// TIA Portal project "4_side_traffic_light_real_clock" (V16)

(* hardware
DEVICE "S7-1200 station_1"  S7-1200 Station
   slot 0: "Rack_0"  S7-1200 Rack  Rack  V1.0
   slot 1: "PLC_1"  CPU 1212C DC/DC/DC  6ES7 212-1AE40-0XB0  V4.4
*)

// ===== PLC "PLC_1"  CPU 1212C DC/DC/DC =====

VAR_GLOBAL   // PLC tag table "Default tag table"
   "Tag_1" AT %M0.0 : Bool;
   "Tag_2" AT %M0.1 : Bool;
   "Tag_3" AT %M0.2 : Bool;
   "green1" AT %Q0.0 : Bool;
   "green2" AT %Q0.1 : Bool;
   "green3" AT %Q0.2 : Bool;
   "green4" AT %Q0.3 : Bool;
   "yellow1" AT %Q0.4 : Bool;
   "yellow2" AT %Q0.5 : Bool;
   "yellow3" AT %Q0.6 : Bool;
   "yellow4" AT %Q0.7 : Bool;
   "red1" AT %Q1.0 : Bool;
   "red2" AT %Q1.1 : Bool;
   "red3" AT %Q1.2 : Bool;
   "red4" AT %Q1.3 : Bool;
   "emergency1" AT %M1.2 : Bool;
   "emergency2" AT %M1.3 : Bool;
   "emergency3" AT %M1.4 : Bool;
   "emergency4" AT %M1.5 : Bool;
   "set date and time" AT %M9.0 : Bool;
   "night mode" AT %M4.3 : Bool;
   "yellow blinker" AT %Q1.6 : Bool;
END_VAR

DATA_BLOCK "read data block"   // DB2
{ S7_Optimized_Access := 'TRUE' }
VERSION : 0.1
   VAR
      "read data block" : DTL;
      status : Int;
   END_VAR
BEGIN
END_DATA_BLOCK

DATA_BLOCK "write data block"   // DB3
{ S7_Optimized_Access := 'TRUE' }
VERSION : 0.1
   VAR
      "write data block" : DTL;
      status : Int;
   END_VAR
BEGIN
END_DATA_BLOCK

// folder: System blocks/Program resources

DATA_BLOCK "timer1"   // DB1
{ S7_Optimized_Access := 'TRUE' }
AUTHOR : Simatic
FAMILY : IEC
NAME : IEC_TMR
VERSION : 1.0
// stored: InstanceOfName IEC_TIMER
"IEC_TIMER"
BEGIN
END_DATA_BLOCK

DATA_BLOCK "timer2"   // DB4
{ S7_Optimized_Access := 'TRUE' }
AUTHOR : Simatic
FAMILY : IEC
NAME : IEC_TMR
VERSION : 1.0
// stored: InstanceOfName IEC_TIMER
"IEC_TIMER"
BEGIN
END_DATA_BLOCK

DATA_BLOCK "timer3"   // DB5
{ S7_Optimized_Access := 'TRUE' }
AUTHOR : Simatic
FAMILY : IEC
NAME : IEC_TMR
VERSION : 1.0
// stored: InstanceOfName IEC_TIMER
"IEC_TIMER"
BEGIN
END_DATA_BLOCK

// folder: (top level)

ORGANIZATION_BLOCK "Main"   // OB1, LAD, ProgramCycle
TITLE = "Main Program Sweep (Cycle)"
{ S7_Optimized_Access := 'TRUE' }
VERSION : 0.1
   VAR_INPUT
      Initial_Call : Bool;   // Initial call of this OB
      Remanence : Bool;   // =True, if remanent data are available
   END_VAR
BEGIN

REGION Network 1
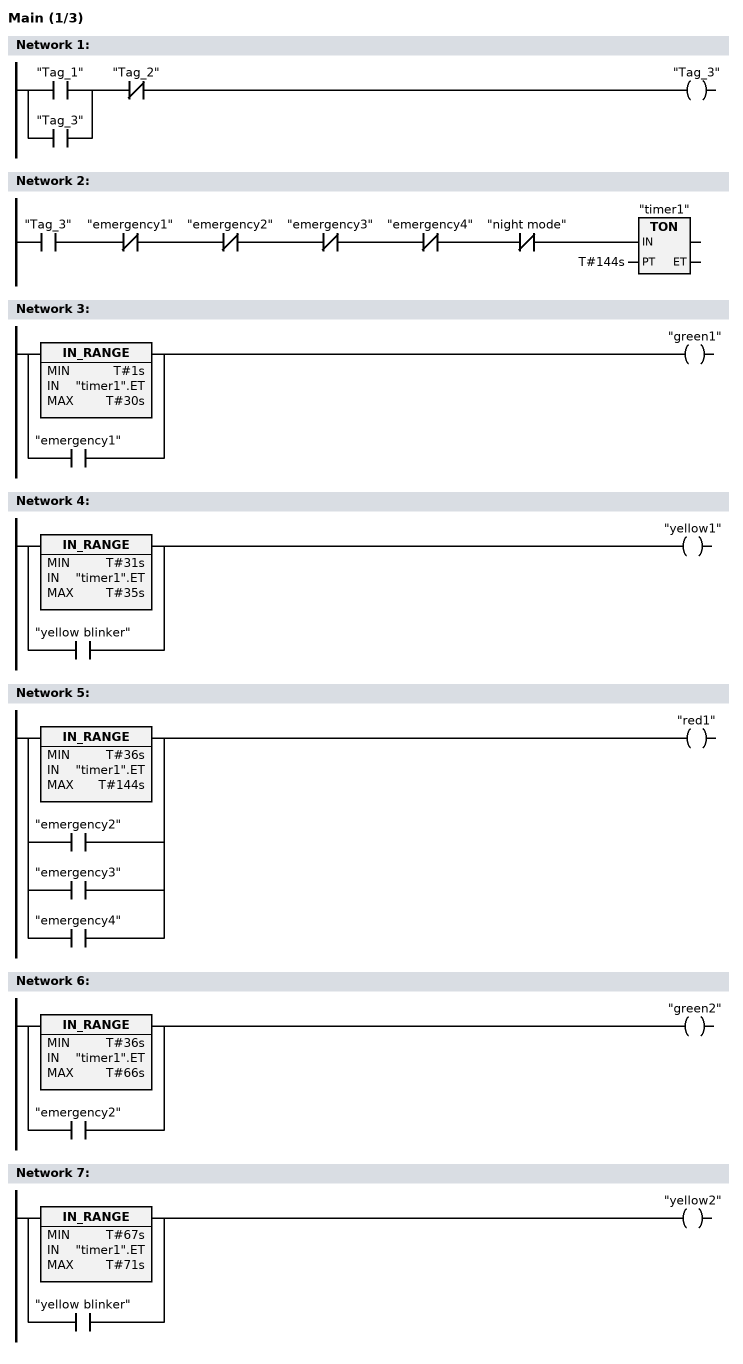
   RUNG wire#powerrail
      Contact( "Tag_1" )
      wire#w1
      I_Contact( "Tag_2" )
      Coil( "Tag_3" )
   END_RUNG
   RUNG wire#powerrail
      Contact( "Tag_3" )
   END_RUNG wire#w1
   // the same network as SCL:
   "Tag_3" := ("Tag_1" OR "Tag_3") AND NOT "Tag_2";
END_REGION

REGION Network 2
   "timer1".TON(IN := "Tag_3" AND NOT "emergency1" AND NOT "emergency2" AND NOT "emergency3" AND NOT "emergency4" AND NOT "night mode",
                PT := T#144s);
END_REGION

REGION Network 3
   RUNG wire#powerrail
      { S7_Templates := "SrcType := DInt" } InRange(min := T#1s, in := "timer1".ET, max := T#30s)
      wire#w1
      Coil( "green1" )
   END_RUNG
   RUNG wire#powerrail
      Contact( "emergency1" )
   END_RUNG wire#w1
   // the same network as SCL:
   "green1" := ((T#1s <= "timer1".ET) AND ("timer1".ET <= T#30s)) OR "emergency1";
END_REGION

REGION Network 4
   RUNG wire#powerrail
      { S7_Templates := "SrcType := DInt" } InRange(min := T#31s, in := "timer1".ET, max := T#35s)
      wire#w1
      Coil( "yellow1" )
   END_RUNG
   RUNG wire#powerrail
      Contact( "yellow blinker" )
   END_RUNG wire#w1
   // the same network as SCL:
   "yellow1" := ((T#31s <= "timer1".ET) AND ("timer1".ET <= T#35s)) OR "yellow blinker";
END_REGION

REGION Network 5
   RUNG wire#powerrail
      { S7_Templates := "SrcType := DInt" } InRange(min := T#36s, in := "timer1".ET, max := T#144s)
      wire#w1
      Coil( "red1" )
   END_RUNG
   RUNG wire#powerrail
      Contact( "emergency2" )
   END_RUNG wire#w1
   RUNG wire#powerrail
      Contact( "emergency3" )
   END_RUNG wire#w1
   RUNG wire#powerrail
      Contact( "emergency4" )
   END_RUNG wire#w1
   // the same network as SCL:
   "red1" := ((T#36s <= "timer1".ET) AND ("timer1".ET <= T#144s)) OR "emergency2" OR "emergency3" OR "emergency4";
END_REGION

REGION Network 6
   RUNG wire#powerrail
      { S7_Templates := "SrcType := DInt" } InRange(min := T#36s, in := "timer1".ET, max := T#66s)
      wire#w1
      Coil( "green2" )
   END_RUNG
   RUNG wire#powerrail
      Contact( "emergency2" )
   END_RUNG wire#w1
   // the same network as SCL:
   "green2" := ((T#36s <= "timer1".ET) AND ("timer1".ET <= T#66s)) OR "emergency2";
END_REGION

REGION Network 7
   RUNG wire#powerrail
      { S7_Templates := "SrcType := DInt" } InRange(min := T#67s, in := "timer1".ET, max := T#71s)
      wire#w1
      Coil( "yellow2" )
   END_RUNG
   RUNG wire#powerrail
      Contact( "yellow blinker" )
   END_RUNG wire#w1
   // the same network as SCL:
   "yellow2" := ((T#67s <= "timer1".ET) AND ("timer1".ET <= T#71s)) OR "yellow blinker";
END_REGION

REGION Network 8
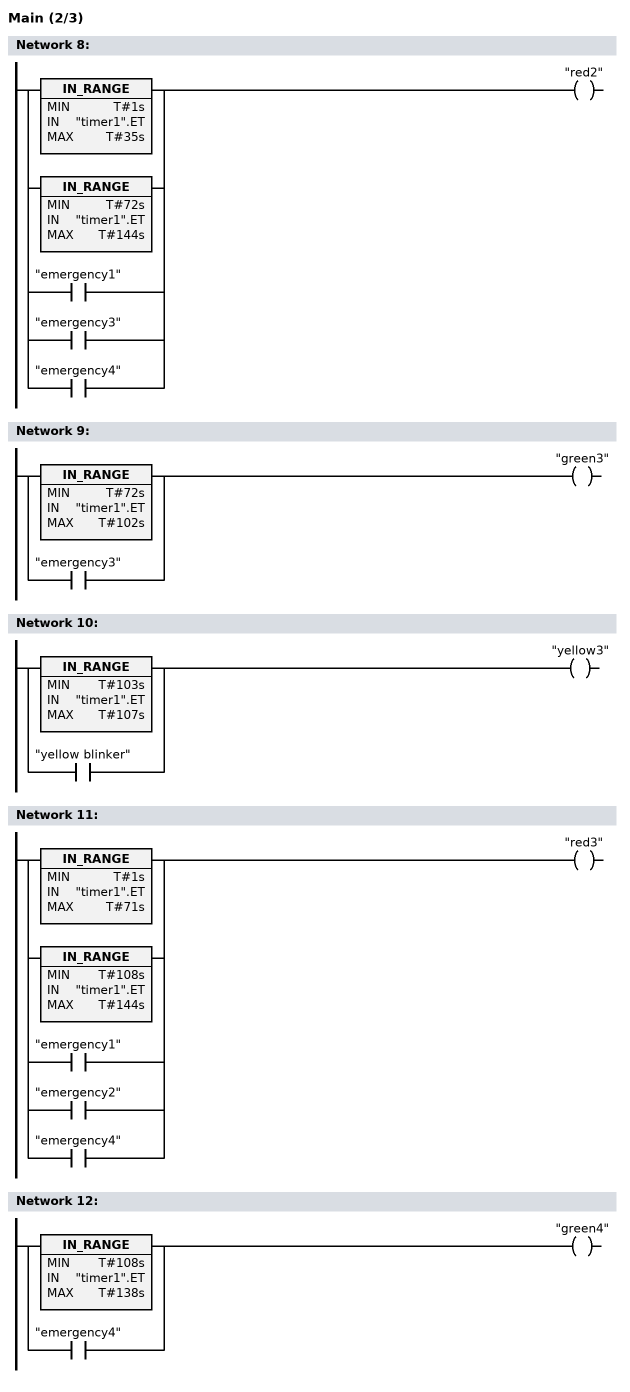
   RUNG wire#powerrail
      { S7_Templates := "SrcType := DInt" } InRange(min := T#1s, in := "timer1".ET, max := T#35s)
      wire#w1
      Coil( "red2" )
   END_RUNG
   RUNG wire#powerrail
      { S7_Templates := "SrcType := DInt" } InRange(min := T#72s, in := "timer1".ET, max := T#144s)
   END_RUNG wire#w1
   RUNG wire#powerrail
      Contact( "emergency1" )
   END_RUNG wire#w1
   RUNG wire#powerrail
      Contact( "emergency3" )
   END_RUNG wire#w1
   RUNG wire#powerrail
      Contact( "emergency4" )
   END_RUNG wire#w1
   // the same network as SCL:
   "red2" := ((T#1s <= "timer1".ET) AND ("timer1".ET <= T#35s)) OR ((T#72s <= "timer1".ET) AND ("timer1".ET <= T#144s)) OR "emergency1" OR "emergency3" OR "emergency4";
END_REGION

REGION Network 9
   RUNG wire#powerrail
      { S7_Templates := "SrcType := DInt" } InRange(min := T#72s, in := "timer1".ET, max := T#102s)
      wire#w1
      Coil( "green3" )
   END_RUNG
   RUNG wire#powerrail
      Contact( "emergency3" )
   END_RUNG wire#w1
   // the same network as SCL:
   "green3" := ((T#72s <= "timer1".ET) AND ("timer1".ET <= T#102s)) OR "emergency3";
END_REGION

REGION Network 10
   RUNG wire#powerrail
      { S7_Templates := "SrcType := DInt" } InRange(min := T#103s, in := "timer1".ET, max := T#107s)
      wire#w1
      Coil( "yellow3" )
   END_RUNG
   RUNG wire#powerrail
      Contact( "yellow blinker" )
   END_RUNG wire#w1
   // the same network as SCL:
   "yellow3" := ((T#103s <= "timer1".ET) AND ("timer1".ET <= T#107s)) OR "yellow blinker";
END_REGION

REGION Network 11
   RUNG wire#powerrail
      { S7_Templates := "SrcType := DInt" } InRange(min := T#1s, in := "timer1".ET, max := T#71s)
      wire#w1
      Coil( "red3" )
   END_RUNG
   RUNG wire#powerrail
      { S7_Templates := "SrcType := DInt" } InRange(min := T#108s, in := "timer1".ET, max := T#144s)
   END_RUNG wire#w1
   RUNG wire#powerrail
      Contact( "emergency1" )
   END_RUNG wire#w1
   RUNG wire#powerrail
      Contact( "emergency2" )
   END_RUNG wire#w1
   RUNG wire#powerrail
      Contact( "emergency4" )
   END_RUNG wire#w1
   // the same network as SCL:
   "red3" := ((T#1s <= "timer1".ET) AND ("timer1".ET <= T#71s)) OR ((T#108s <= "timer1".ET) AND ("timer1".ET <= T#144s)) OR "emergency1" OR "emergency2" OR "emergency4";
END_REGION

REGION Network 12
   RUNG wire#powerrail
      { S7_Templates := "SrcType := DInt" } InRange(min := T#108s, in := "timer1".ET, max := T#138s)
      wire#w1
      Coil( "green4" )
   END_RUNG
   RUNG wire#powerrail
      Contact( "emergency4" )
   END_RUNG wire#w1
   // the same network as SCL:
   "green4" := ((T#108s <= "timer1".ET) AND ("timer1".ET <= T#138s)) OR "emergency4";
END_REGION

REGION Network 13
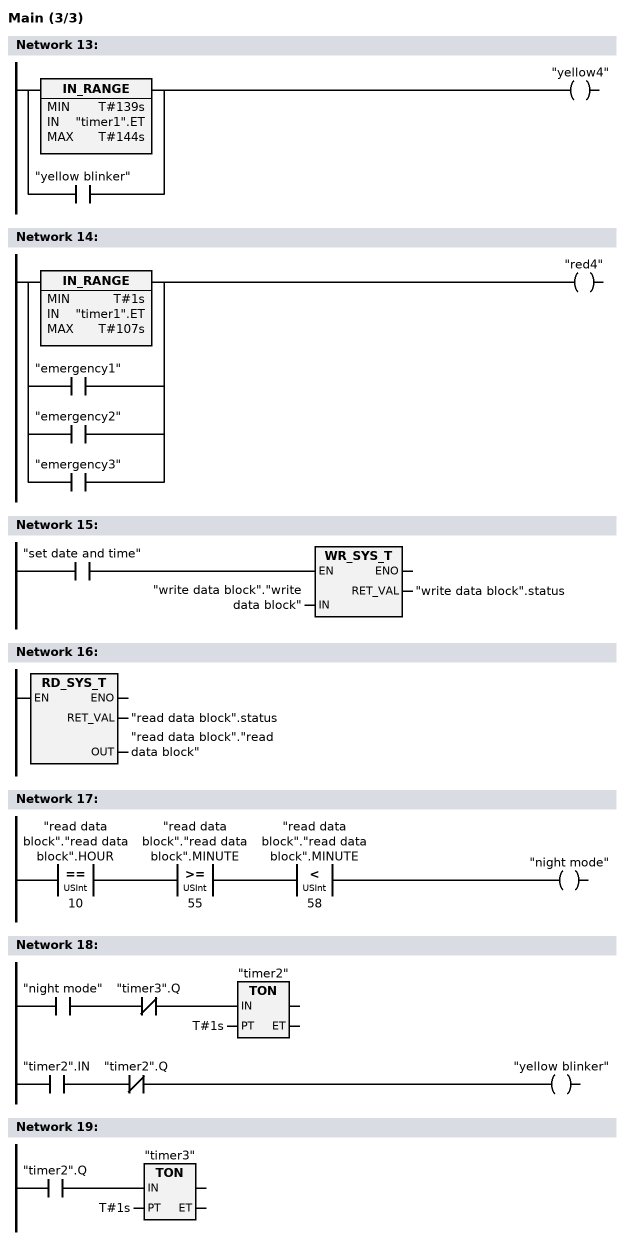
   RUNG wire#powerrail
      { S7_Templates := "SrcType := DInt" } InRange(min := T#139s, in := "timer1".ET, max := T#144s)
      wire#w1
      Coil( "yellow4" )
   END_RUNG
   RUNG wire#powerrail
      Contact( "yellow blinker" )
   END_RUNG wire#w1
   // the same network as SCL:
   "yellow4" := ((T#139s <= "timer1".ET) AND ("timer1".ET <= T#144s)) OR "yellow blinker";
END_REGION

REGION Network 14
   RUNG wire#powerrail
      { S7_Templates := "SrcType := DInt" } InRange(min := T#1s, in := "timer1".ET, max := T#107s)
      wire#w1
      Coil( "red4" )
   END_RUNG
   RUNG wire#powerrail
      Contact( "emergency1" )
   END_RUNG wire#w1
   RUNG wire#powerrail
      Contact( "emergency2" )
   END_RUNG wire#w1
   RUNG wire#powerrail
      Contact( "emergency3" )
   END_RUNG wire#w1
   // the same network as SCL:
   "red4" := ((T#1s <= "timer1".ET) AND ("timer1".ET <= T#107s)) OR "emergency1" OR "emergency2" OR "emergency3";
END_REGION

REGION Network 15
   IF "set date and time" THEN
       "write data block".status := WR_SYS_T(IN := "write data block"."write data block");
   END_IF;
END_REGION

REGION Network 16
   "read data block".status := RD_SYS_T(OUT => "read data block"."read data block");
END_REGION

REGION Network 17
   RUNG wire#powerrail
      { S7_Templates := "SrcType := USInt" } EQ_Contact(in1 := "read data block"."read data block".HOUR, in2 := 10)
      { S7_Templates := "SrcType := USInt" } GE_Contact(in1 := "read data block"."read data block".MINUTE, in2 := 55)
      { S7_Templates := "SrcType := USInt" } LT_Contact(in1 := "read data block"."read data block".MINUTE, in2 := 58)
      Coil( "night mode" )
   END_RUNG
   // the same network as SCL:
   "night mode" := ("read data block"."read data block".HOUR = 10) AND ("read data block"."read data block".MINUTE >= 55) AND ("read data block"."read data block".MINUTE < 58);
END_REGION

REGION Network 18
   "timer2".TON(IN := "night mode" AND NOT "timer3".Q, PT := T#1s);
   "yellow blinker" := "timer2".IN AND NOT "timer2".Q;
END_REGION

REGION Network 19
   "timer3".TON(IN := "timer2".Q, PT := T#1s);
END_REGION
END_ORGANIZATION_BLOCK